// TIA Portal V20 export
TYPE "LConSMC_typeStopDynamics"
// [Einheit der Achse] Dynamiken zum Stoppen der Achse  Wirksam wenn "enable" = FALSE oder wenn "speedMatch" = FALSE bei laufender Bahn / [Unit of the axis] Dynamics for stopping the axis  Active if "enable" = FALSE or "speedMatch" = FLASE and running web
// stored: Access Published
   STRUCT
      deceleration : Real := -1.0;   // Verzögerung in Achseinheit / Deceleration value: Units are taken from the TO
      jerk : Real := -1.0;   // Ruckbegrenzung in Achseinheit / Jerk value : Units are taken from the TO
      abortAcceleration : Bool := FALSE;   // TRUE: Setze aktuelle Beschleunigung auf 0 FALSE: Baue aktuelle Beschleunigung über konfigurierten Ruck ab / TRUE: Abort acceleration immediately, FALSE: Reduce current acceleration via Jerk
   END_STRUCT;
END_TYPE
